PROGRAM P_Inputs
VAR
	fbJoystickWinch 				: FB_JoystickInputScaling;
	fbJoystickCyl 					: FB_JoystickInputScaling;
	fbWinchPosition 				: FB_Encoder;
	fbCylPistonPosition 			: FB_AnalogInputScaling;
	fbPressureSupply 				: FB_AnalogInputScaling;
	fbPressureReturn 				: FB_AnalogInputScaling;
	fbPressureCyl_A_PistonSide 		: FB_AnalogInputScaling;
	fbPressureCyl_B_RodSide			: FB_AnalogInputScaling;
	fbPressureWinch_A_Input 		: FB_AnalogInputScaling;
	fbPressureWinch_A1_Input 		: FB_AnalogInputScaling;
	fbPressureWinch_B_Output		: FB_AnalogInputScaling;
	fbPressureWinch_B1_Output		: FB_AnalogInputScaling;
	fbPressureWinchDrain			: FB_AnalogInputScaling;
	fbFlowWinch						: FB_FlowMeterInputScaling;
	
	
	
END_VAR

fbJoystickWinch(
	bEnable := G_Work.bManualMode,
	nRawInput := G_Inputs.stJoyY.nValue,
	stJoystickInputScaling := G_Parameters.stParam.stJoystickInputScalingY,
	fNormalizedOutput => G_Sensors.fJoystickNormalizedY
);

fbJoystickCyl(
	bEnable := G_Work.bManualMode,
	nRawInput := G_Inputs.stJoyX.nValue,
	stJoystickInputScaling := G_Parameters.stParam.stJoystickInputScalingX,
	fNormalizedOutput => G_Sensors.fJoystickNormalizedX
);

fbWinchPosition (
nRawInput := G_Inputs.nEncoderValue, 
fPosition => G_Sensors.fWinchEncoderPosition,
);

G_Sensors.fWinchWirePosition := fbWinchPosition.fPosition*G_Parameters.stParam.fWinchDrumScaling;

fbCylPistonPosition(
	nRawInput := G_Inputs.stPositionCylPiston.nValue,
	stAnalogInputScaling := G_Parameters.stParam.stCylPistonPositionScaling,
	fOutput => G_Sensors.fPositionCylPiston
);

fbPressureSupply(
	nRawInput := G_Inputs.stPressureSupply.nValue,
	stAnalogInputScaling := G_Parameters.stParam.stPressureSensorScaling400bar,
	fOutput => G_Sensors.fPressureSupply
);

fbPressureReturn(
	nRawInput := G_Inputs.stPressureReturn.nValue,
	stAnalogInputScaling := G_Parameters.stParam.stPressureSensorScaling40bar,
	fOutput => G_Sensors.fPressureReturn
);

fbPressureCyl_A_PistonSide(
	nRawInput := G_Inputs.stPressureCyl_A_PistonSide.nValue,
	stAnalogInputScaling := G_Parameters.stParam.stPressureSensorScaling400bar,
	fOutput => G_Sensors.fPressureCyl_A_PistonSide
);

fbPressureCyl_B_RodSide(
	nRawInput := G_Inputs.stPressureCyl_B_RodSide.nValue,
	stAnalogInputScaling := G_Parameters.stParam.stPressureSensorScaling400bar,
	fOutput => G_Sensors.fPressureCyl_B_RodSide
);

fbPressureWinch_A_Input(
	nRawInput := G_Inputs.stPressureWinch_A_Input.nValue,
	stAnalogInputScaling := G_Parameters.stParam.stPressureSensorScaling400bar,
	fOutput => G_Sensors.fPressureWinch_A_Input
);

fbPressureWinch_A1_Input(
	nRawInput := G_Inputs.stPressureWinch_A1_Input.nValue,
	stAnalogInputScaling := G_Parameters.stParam.stPressureSensorScaling400bar,
	fOutput => G_Sensors.fPressureWinch_A1_Side
);

fbPressureWinch_B_Output(
	nRawInput := G_Inputs.stPressureWinch_B_Output.nValue,
	stAnalogInputScaling := G_Parameters.stParam.stPressureSensorScaling400bar,
	fOutput => G_Sensors.fPressureWinch_B_Output
);

fbPressureWinch_B1_Output(
	nRawInput := G_Inputs.stPressureWinch_B1_Output.nValue,
	stAnalogInputScaling := G_Parameters.stParam.stPressureSensorScaling400bar,
	fOutput => G_Sensors.fPressureWinch_B1_Output
);

fbPressureWinchDrain(
	nRawInput := G_Inputs.stPressureWinchDrain.nValue,
	stAnalogInputScaling := G_Parameters.stParam.stPressureSensorScaling40bar,
	fOutput => G_Sensors.fPressureWinchDrain
);

fbFlowWinch(
	nRawInput := G_Inputs.stFlowWinch.nValue,
	stFlowMeterInputScaling := G_Parameters.stParam.stFlowMeterInputScaling,
	fNormalizedOutput => G_Sensors.fWinchFlow
);

END_PROGRAM

(* stored: Version 1.1.0.1, ProductVersion 3.1.4024.11
   POU P_Inputs: Id {8b676dbd-393f-42d6-8803-330b6e90ab14}, SpecialFunc None *)
